FUNCTION_BLOCK IW (* Input service interface function block for word input data *)
  (* Description: Copyright (c) 2015, 2016 fortiss GmbH This program and the accompanying materials are made available under the terms of the Eclipse Public License 2.0 which is available at https://www.eclipse.org/legal/epl-2.0/ SPDX-License-Identifier: EPL-2.0 *)
  (* Version 3.0, 2025-04-14, Patrick Aigner, changed package *)
  (* Version 1.1, 2016-07-18, Alois Zoitl, fortiss GmbH *)
  (* Version 1.0, 2015-09-22, Gerd Kainz, fortiss GmbH *)
  PACKAGE eclipse4diac::io;
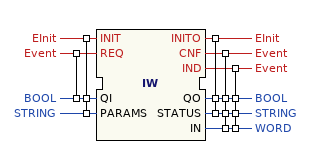
  EVENT_INPUT
    INIT : EInit WITH QI, PARAMS; (* Service Initialization *)
    REQ WITH QI; (* Service Request *)
  END_EVENT
  EVENT_OUTPUT
    INITO : EInit WITH QO, STATUS; (* Initialization Confirm *)
    CNF WITH QO, STATUS, IN; (* Confirmation of Requested Service *)
    IND WITH QO, STATUS, IN; (* Indication from Resource *)
  END_EVENT
  VAR_INPUT
    QI : BOOL; (* Event Input Qualifier *)
    PARAMS : STRING; (* Service Parameters *)
  END_VAR
  VAR_OUTPUT
    QO : BOOL; (* Event Output Qualifier *)
    STATUS : STRING; (* Service Status *)
    IN : WORD; (* Input data from resource *)
  END_VAR
END_FUNCTION_BLOCK
